Yaskawa INFORM job: TEST-GET-DATA.JBI

/JOB
//NAME TEST-GET-DATA
//POS
///NPOS 0,0,0,0,0,0
//INST
///DATE 2018/08/30 09:27
///ATTR SC,RW
///GROUP1 RB1
NOP
MACRO1 MJ#(1) ARGF1 ARGF71
PAUSE
MACRO1 MJ#(2) ARGF10 ARGF70
END
